PROGRAM MAIN
VAR
END_VAR

// PRUEBA PARA EL MAIN EN LUGAR DEL MASTER//

//no jala //
// primer cosa ///

//main//

END_PROGRAM

(* stored: Version 1.1.0.1, ProductVersion 3.1.4024.9
   POU MAIN: Id {a1e7293a-1635-4c1b-8f12-114f4e7f9a94}, SpecialFunc None *)
